Universal Robots PolyScope program: RC_E4_PICK_420.urp

Program RC_E4_PICK_420 (createdIn=3.0.0 lastSavedIn=3.0.0 directory=/programs installation=default)
Robot Program (runOnlyOnce=true motionType=MoveJ speed=1.047198 acceleration=1.396263 useActiveTCP=false)
  'Program generated by RoboDK v4.1.0 for UR3e_HORNO on 27/07/2022 12:06:32'
  'Using nominal kinematics.'
  'Using Ref. Frame Inspeccion 02: p[-0.386000, 0.280000, -0.011500, 0.000000, 0.000000, 0.000000]'
  'Using TCP 0208-0001-0001-307-000-3 Horno: p[0.000000, 0.000000, 0.038000, 0.000000, 0.000000, 0.000000]'
  Script: set_tcp(p[0.000000, 0.000000, 0.038000, 0.000000, 0.000000, 0.000000])
  Script: movej([3.161315, -1.272520, -1.014385, -0.852593, -0.017453, 0.000000],0.60000,0.12500,0,0.0000)
  Script: movej([3.161315, -1.892354, -2.373425, 1.125932, 0.000000, 0.000000],0.60000,0.12500,0,0.0000)
  Script: movej([3.153927, -2.488789, -1.856352, 1.205290, 1.568243, 0.000019],0.60000,0.12500,0,0.0000)
  Script: movej([3.011344, -2.548727, -1.716896, 1.143166, 1.727401, -0.035605],0.60000,0.12500,0,0.0000)
  Script: movej([3.343368, -2.486848, -1.938955, 1.303406, 1.395438, -0.041939],0.60000,0.12500,0,0.0000)
  Script: movej([3.011344, -2.548727, -1.716896, 1.143166, 1.727401, -0.035605],0.60000,0.12500,0,0.0000)
  Script: movej([2.954915, -2.448996, -2.145047, 1.471788, 1.783820, -0.034501],0.60000,0.12500,0,0.0000)
  Script: movej([3.458409, -2.458919, -2.431228, 1.768281, 1.280418, -0.044239],0.60000,0.12500,0,0.0000)
  Script: movej([3.161315, -1.892354, -2.373425, 1.125932, 0.000000, 0.000000],0.60000,0.12500,0,0.0000)
  Script: movej([3.161315, -1.892354, -2.373425, 1.125932, 0.000000, 0.000000],0.60000,0.12500,0,0.0000)
  Script: movej([3.161315, -1.272520, -1.014385, -0.852593, -0.017453, 0.000000],0.60000,0.12500,0,0.0000)
